(* PLC project Beremiz Direct Raw Ethernet Study PLC, Study Stand Beremiz Direct Raw PLC 1 *)
(* stored: creationDateTime 2026-06-15T12:00:00, modificationDateTime 2026-06-15T12:00:00 *)

PROGRAM plc_prg
  VAR_EXTERNAL
    RawSensorValue : UINT;
    RawThreshold : UINT;
    RawForcedOutput : UINT;
    RawSequence : UDINT;
    RawOutputCommand : UINT;
  END_VAR
  VAR
    sensor_value : UINT;
    threshold : UINT;
    remote_output_echo : UINT;
    sequence : UDINT;
    alarm : BOOL;
    output_command : UINT;
  END_VAR

            sensor_value := RawSensorValue;
threshold := RawThreshold;
remote_output_echo := RawForcedOutput;
sequence := RawSequence;

alarm := sensor_value > threshold;

IF alarm THEN
    output_command := UINT#1;
ELSE
    output_command := UINT#0;
END_IF;

RawOutputCommand := output_command;
          
END_PROGRAM

CONFIGURATION config
  RESOURCE resource1 ON PLC
    TASK task0(INTERVAL := T#100ms, PRIORITY := 0);
    PROGRAM instance0 WITH task0 : plc_prg;
  END_RESOURCE
END_CONFIGURATION
